// TIA Portal V18 export
TYPE "LGasp_typeHMI_DS"
// stored: IsFailsafeCompliant false
   STRUCT
      val : LReal;
      ll : LReal;
      hl : LReal;
   END_STRUCT;
END_TYPE
